Xinje XDPPro project, PLC1: XD3-32 (software 3.7.14 2021-12-24)

PROGRAM 梯形图

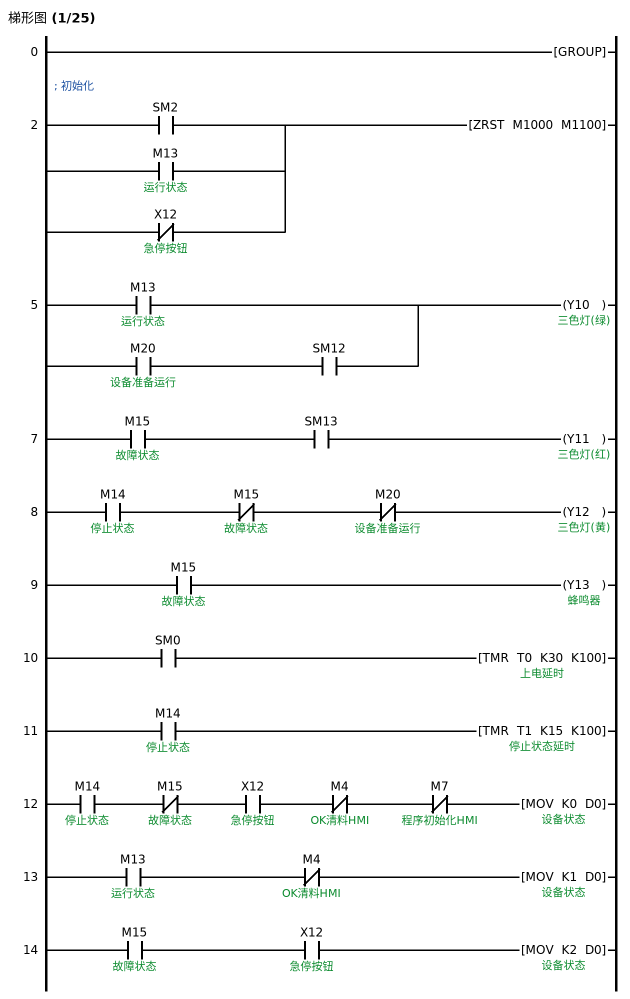
GROUP
; 初始化
LD     SM2
OR     M13	; 运行状态
ORI    X12	; 急停按钮
ZRST   M1000 M1100
LD     M13	; 运行状态
LD     M20	; 设备准备运行
AND    SM12
ORB
OUT    Y10	; 三色灯(绿)
LD     M15	; 故障状态
AND    SM13
OUT    Y11	; 三色灯(红)
LD     M14	; 停止状态
ANI    M15	; 故障状态
ANI    M20	; 设备准备运行
OUT    Y12	; 三色灯(黄)
LD     M15	; 故障状态
OUT    Y13	; 蜂鸣器
LD     SM0
TMR    T0 K30 K100	; 上电延时
LD     M14	; 停止状态
TMR    T1 K15 K100	; 停止状态延时
LD     M14	; 停止状态
ANI    M15	; 故障状态
AND    X12	; 急停按钮
ANI    M4	; OK清料HMI
ANI    M7	; 程序初始化HMI
MOV    K0 D0	; 设备状态
LD     M13	; 运行状态
ANI    M4	; OK清料HMI
MOV    K1 D0	; 设备状态
LD     M15	; 故障状态
AND    X12	; 急停按钮
MOV    K2 D0	; 设备状态

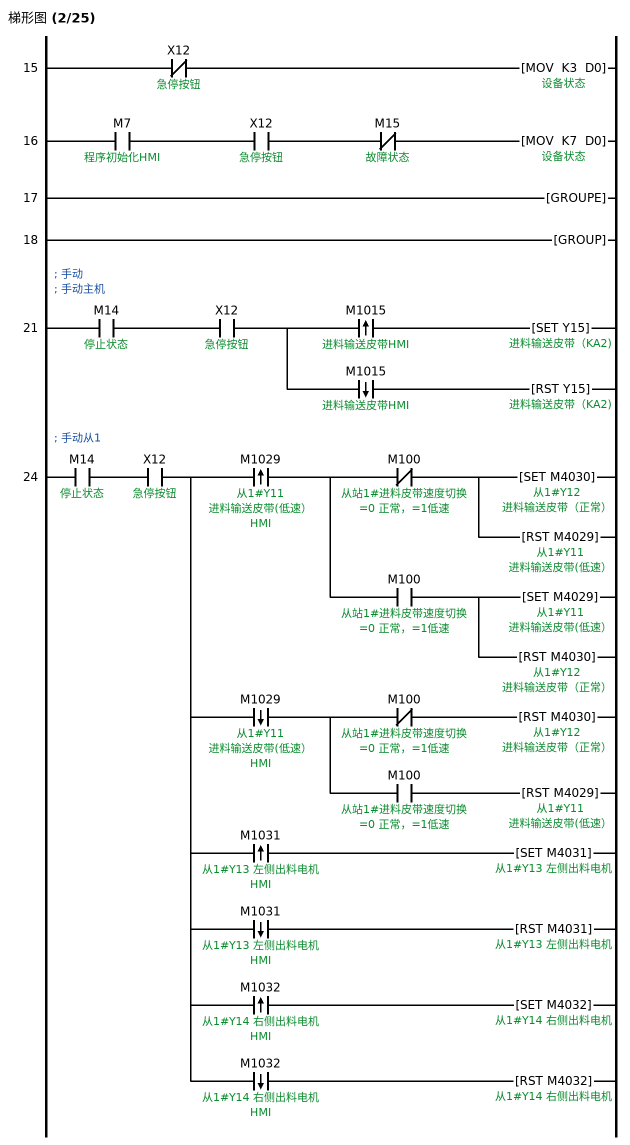
LDI    X12	; 急停按钮
MOV    K3 D0	; 设备状态
LD     M7	; 程序初始化HMI
AND    X12	; 急停按钮
ANI    M15	; 故障状态
MOV    K7 D0	; 设备状态
GROUPE
GROUP
; 手动
; 手动主机
LD     M14	; 停止状态
AND    X12	; 急停按钮
MPS
ANDP   M1015	; 进料输送皮带HMI
SET    Y15	; 进料输送皮带（KA2)
MPP
ANDF   M1015	; 进料输送皮带HMI
RST    Y15	; 进料输送皮带（KA2)
; 手动从1
LD     M14	; 停止状态
AND    X12	; 急停按钮
MPS
ANDP   M1029	; 从1#Y11 进料输送皮带(低速）       HMI
MPS
ANI    M100	; 从站1#进料皮带速度切换=0 正常，=1低速
SET    M4030	; 从1#Y12 进料输送皮带（正常）
RST    M4029	; 从1#Y11 进料输送皮带(低速）
MPP
AND    M100	; 从站1#进料皮带速度切换=0 正常，=1低速
SET    M4029	; 从1#Y11 进料输送皮带(低速）
RST    M4030	; 从1#Y12 进料输送皮带（正常）
MRD
ANDF   M1029	; 从1#Y11 进料输送皮带(低速）       HMI
MPS
ANI    M100	; 从站1#进料皮带速度切换=0 正常，=1低速
RST    M4030	; 从1#Y12 进料输送皮带（正常）
MPP
AND    M100	; 从站1#进料皮带速度切换=0 正常，=1低速
RST    M4029	; 从1#Y11 进料输送皮带(低速）
MRD
ANDP   M1031	; 从1#Y13 左侧出料电机       HMI
SET    M4031	; 从1#Y13 左侧出料电机
MRD
ANDF   M1031	; 从1#Y13 左侧出料电机       HMI
RST    M4031	; 从1#Y13 左侧出料电机
MRD
ANDP   M1032	; 从1#Y14 右侧出料电机       HMI
SET    M4032	; 从1#Y14 右侧出料电机
MPP
ANDF   M1032	; 从1#Y14 右侧出料电机       HMI
RST    M4032	; 从1#Y14 右侧出料电机

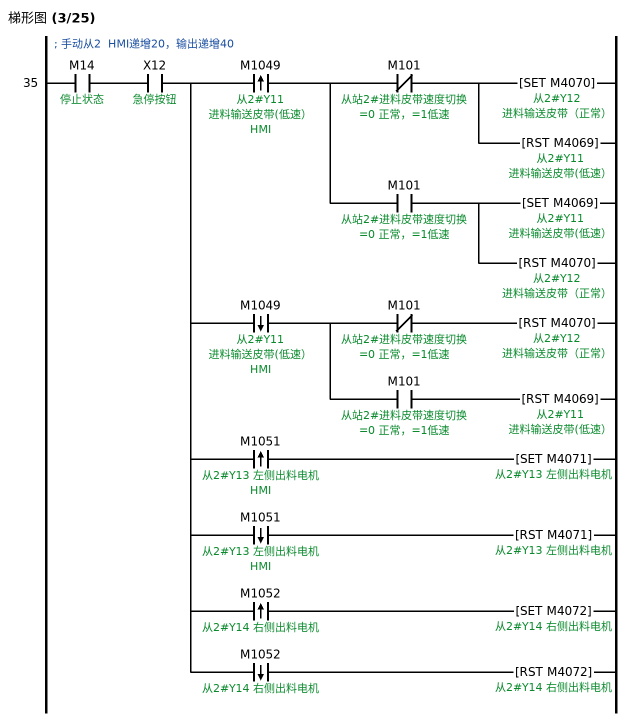
; 手动从2  HMI递增20，输出递增40
LD     M14	; 停止状态
AND    X12	; 急停按钮
MPS
ANDP   M1049	; 从2#Y11 进料输送皮带(低速）       HMI
MPS
ANI    M101	; 从站2#进料皮带速度切换=0 正常，=1低速
SET    M4070	; 从2#Y12 进料输送皮带（正常）
RST    M4069	; 从2#Y11 进料输送皮带(低速）
MPP
AND    M101	; 从站2#进料皮带速度切换=0 正常，=1低速
SET    M4069	; 从2#Y11 进料输送皮带(低速）
RST    M4070	; 从2#Y12 进料输送皮带（正常）
MRD
ANDF   M1049	; 从2#Y11 进料输送皮带(低速）       HMI
MPS
ANI    M101	; 从站2#进料皮带速度切换=0 正常，=1低速
RST    M4070	; 从2#Y12 进料输送皮带（正常）
MPP
AND    M101	; 从站2#进料皮带速度切换=0 正常，=1低速
RST    M4069	; 从2#Y11 进料输送皮带(低速）
MRD
ANDP   M1051	; 从2#Y13 左侧出料电机       HMI
SET    M4071	; 从2#Y13 左侧出料电机
MRD
ANDF   M1051	; 从2#Y13 左侧出料电机       HMI
RST    M4071	; 从2#Y13 左侧出料电机
MRD
ANDP   M1052	; 从2#Y14 右侧出料电机
SET    M4072	; 从2#Y14 右侧出料电机
MPP
ANDF   M1052	; 从2#Y14 右侧出料电机
RST    M4072	; 从2#Y14 右侧出料电机

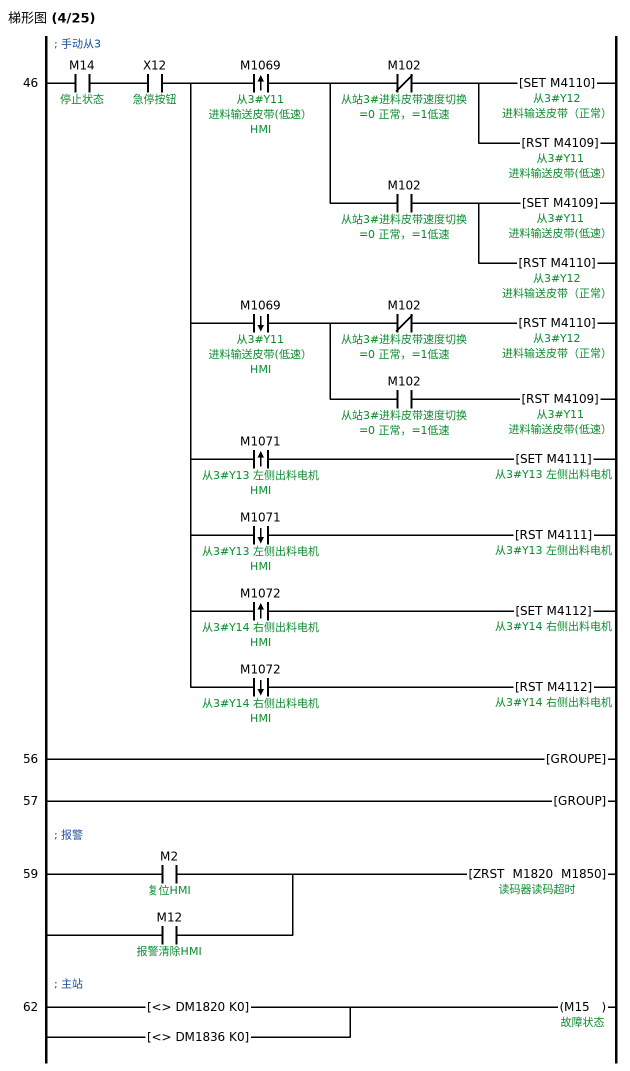
; 手动从3
LD     M14	; 停止状态
AND    X12	; 急停按钮
MPS
ANDP   M1069	; 从3#Y11 进料输送皮带(低速）       HMI
MPS
ANI    M102	; 从站3#进料皮带速度切换=0 正常，=1低速
SET    M4110	; 从3#Y12 进料输送皮带（正常）
RST    M4109	; 从3#Y11 进料输送皮带(低速）
MPP
AND    M102	; 从站3#进料皮带速度切换=0 正常，=1低速
SET    M4109	; 从3#Y11 进料输送皮带(低速）
RST    M4110	; 从3#Y12 进料输送皮带（正常）
MRD
ANDF   M1069	; 从3#Y11 进料输送皮带(低速）       HMI
MPS
ANI    M102	; 从站3#进料皮带速度切换=0 正常，=1低速
RST    M4110	; 从3#Y12 进料输送皮带（正常）
MPP
AND    M102	; 从站3#进料皮带速度切换=0 正常，=1低速
RST    M4109	; 从3#Y11 进料输送皮带(低速）
MRD
ANDP   M1071	; 从3#Y13 左侧出料电机       HMI
SET    M4111	; 从3#Y13 左侧出料电机
MRD
ANDF   M1071	; 从3#Y13 左侧出料电机       HMI
RST    M4111	; 从3#Y13 左侧出料电机
MRD
ANDP   M1072	; 从3#Y14 右侧出料电机       HMI
SET    M4112	; 从3#Y14 右侧出料电机
MPP
ANDF   M1072	; 从3#Y14 右侧出料电机       HMI
RST    M4112	; 从3#Y14 右侧出料电机
GROUPE
GROUP
; 报警
LD     M2	; 复位HMI
OR     M12	; 报警清除HMI
ZRST   M1820 M1850	; 读码器读码超时
; 主站
LD<>   DM1820 K0
OR<>   DM1836 K0
OUT    M15	; 故障状态

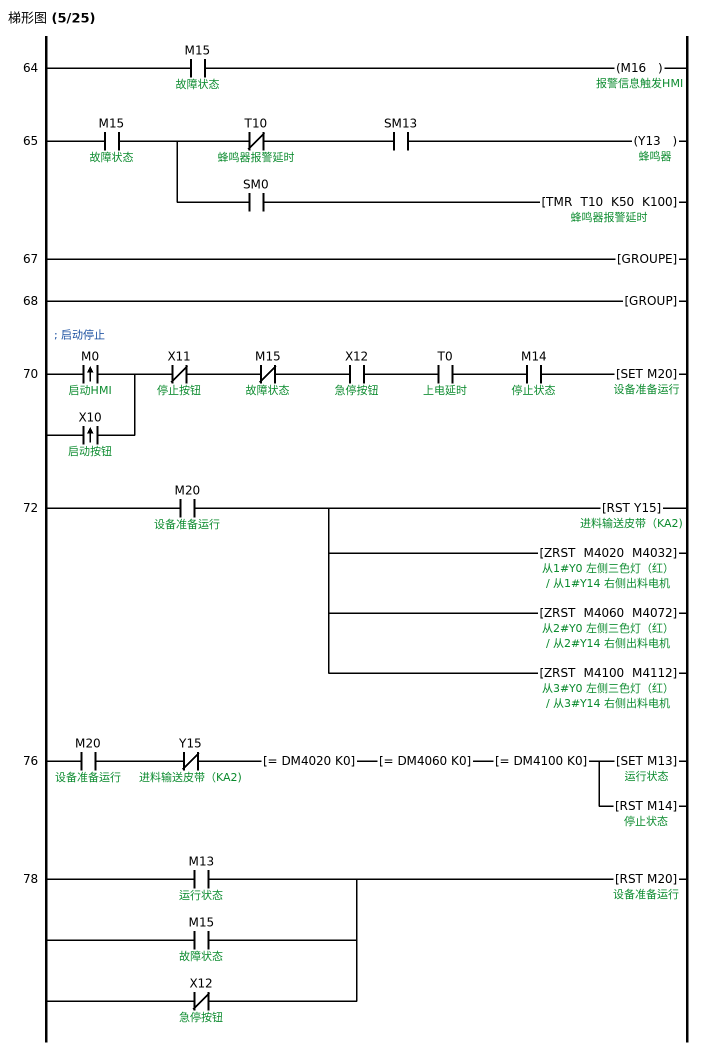
LD     M15	; 故障状态
OUT    M16	; 报警信息触发HMI
LD     M15	; 故障状态
MPS
ANI    T10	; 蜂鸣器报警延时
AND    SM13
OUT    Y13	; 蜂鸣器
MPP
AND    SM0
TMR    T10 K50 K100	; 蜂鸣器报警延时
GROUPE
GROUP
; 启动停止
LDP    M0	; 启动HMI
ORP    X10	; 启动按钮
ANI    X11	; 停止按钮
ANI    M15	; 故障状态
AND    X12	; 急停按钮
AND    T0	; 上电延时
AND    M14	; 停止状态
SET    M20	; 设备准备运行
LD     M20	; 设备准备运行
RST    Y15	; 进料输送皮带（KA2)
ZRST   M4020 M4032	; 从1#Y0 左侧三色灯（红） / 从1#Y14 右侧出料电机
ZRST   M4060 M4072	; 从2#Y0 左侧三色灯（红） / 从2#Y14 右侧出料电机
ZRST   M4100 M4112	; 从3#Y0 左侧三色灯（红） / 从3#Y14 右侧出料电机
LD     M20	; 设备准备运行
ANI    Y15	; 进料输送皮带（KA2)
AND=   DM4020 K0
AND=   DM4060 K0
AND=   DM4100 K0
SET    M13	; 运行状态
RST    M14	; 停止状态
LD     M13	; 运行状态
OR     M15	; 故障状态
ORI    X12	; 急停按钮
RST    M20	; 设备准备运行

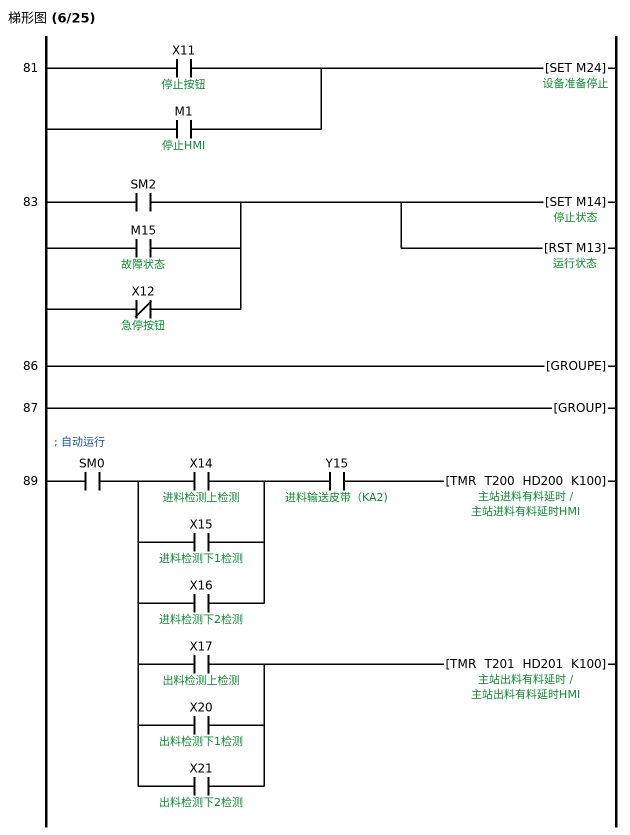
LD     X11	; 停止按钮
OR     M1	; 停止HMI
SET    M24	; 设备准备停止
LD     SM2
OR     M15	; 故障状态
ORI    X12	; 急停按钮
SET    M14	; 停止状态
RST    M13	; 运行状态
GROUPE
GROUP
; 自动运行
LD     SM0
MPS
LD     X14	; 进料检测上检测
OR     X15	; 进料检测下1检测
OR     X16	; 进料检测下2检测
ANB
AND    Y15	; 进料输送皮带（KA2)
TMR    T200 HD200 K100	; 主站进料有料延时 / 主站进料有料延时HMI
MPP
LD     X17	; 出料检测上检测
OR     X20	; 出料检测下1检测
OR     X21	; 出料检测下2检测
ANB
TMR    T201 HD201 K100	; 主站出料有料延时 / 主站出料有料延时HMI

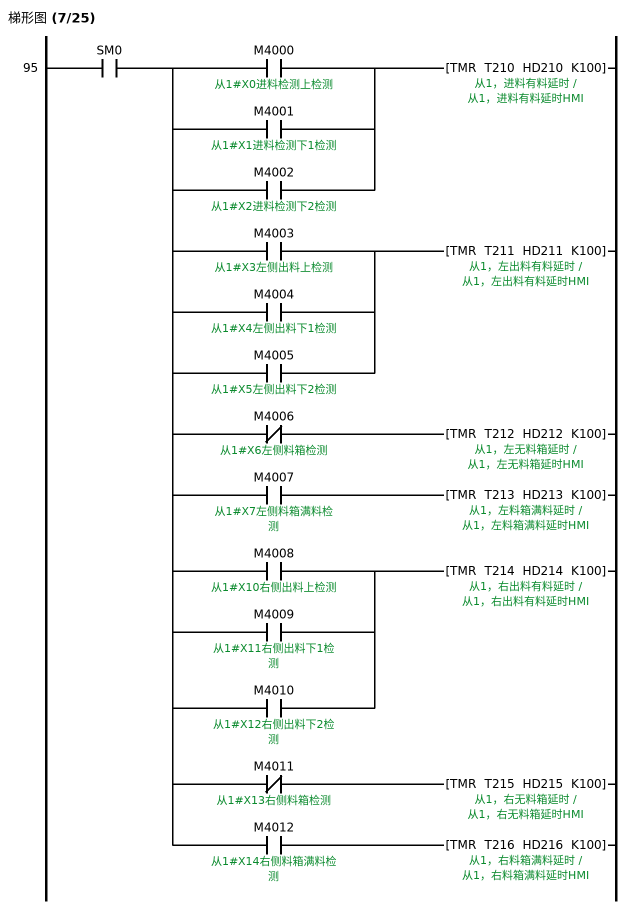
LD     SM0
MPS
LD     M4000	; 从1#X0进料检测上检测
OR     M4001	; 从1#X1进料检测下1检测
OR     M4002	; 从1#X2进料检测下2检测
ANB
TMR    T210 HD210 K100	; 从1，进料有料延时 / 从1，进料有料延时HMI
MRD
LD     M4003	; 从1#X3左侧出料上检测
OR     M4004	; 从1#X4左侧出料下1检测
OR     M4005	; 从1#X5左侧出料下2检测
ANB
TMR    T211 HD211 K100	; 从1，左出料有料延时 / 从1，左出料有料延时HMI
MRD
ANI    M4006	; 从1#X6左侧料箱检测
TMR    T212 HD212 K100	; 从1，左无料箱延时 / 从1，左无料箱延时HMI
MRD
AND    M4007	; 从1#X7左侧料箱满料检测
TMR    T213 HD213 K100	; 从1，左料箱满料延时 / 从1，左料箱满料延时HMI
MRD
LD     M4008	; 从1#X10右侧出料上检测
OR     M4009	; 从1#X11右侧出料下1检测
OR     M4010	; 从1#X12右侧出料下2检测
ANB
TMR    T214 HD214 K100	; 从1，右出料有料延时 / 从1，右出料有料延时HMI
MRD
ANI    M4011	; 从1#X13右侧料箱检测
TMR    T215 HD215 K100	; 从1，右无料箱延时 / 从1，右无料箱延时HMI
MPP
AND    M4012	; 从1#X14右侧料箱满料检测
TMR    T216 HD216 K100	; 从1，右料箱满料延时 / 从1，右料箱满料延时HMI

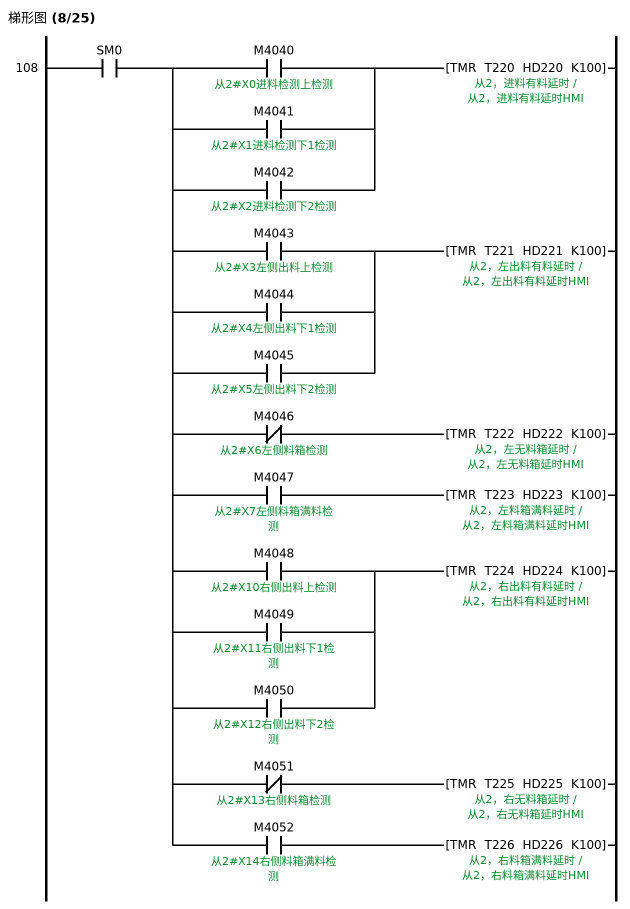
LD     SM0
MPS
LD     M4040	; 从2#X0进料检测上检测
OR     M4041	; 从2#X1进料检测下1检测
OR     M4042	; 从2#X2进料检测下2检测
ANB
TMR    T220 HD220 K100	; 从2，进料有料延时 / 从2，进料有料延时HMI
MRD
LD     M4043	; 从2#X3左侧出料上检测
OR     M4044	; 从2#X4左侧出料下1检测
OR     M4045	; 从2#X5左侧出料下2检测
ANB
TMR    T221 HD221 K100	; 从2，左出料有料延时 / 从2，左出料有料延时HMI
MRD
ANI    M4046	; 从2#X6左侧料箱检测
TMR    T222 HD222 K100	; 从2，左无料箱延时 / 从2，左无料箱延时HMI
MRD
AND    M4047	; 从2#X7左侧料箱满料检测
TMR    T223 HD223 K100	; 从2，左料箱满料延时 / 从2，左料箱满料延时HMI
MRD
LD     M4048	; 从2#X10右侧出料上检测
OR     M4049	; 从2#X11右侧出料下1检测
OR     M4050	; 从2#X12右侧出料下2检测
ANB
TMR    T224 HD224 K100	; 从2，右出料有料延时 / 从2，右出料有料延时HMI
MRD
ANI    M4051	; 从2#X13右侧料箱检测
TMR    T225 HD225 K100	; 从2，右无料箱延时 / 从2，右无料箱延时HMI
MPP
AND    M4052	; 从2#X14右侧料箱满料检测
TMR    T226 HD226 K100	; 从2，右料箱满料延时 / 从2，右料箱满料延时HMI

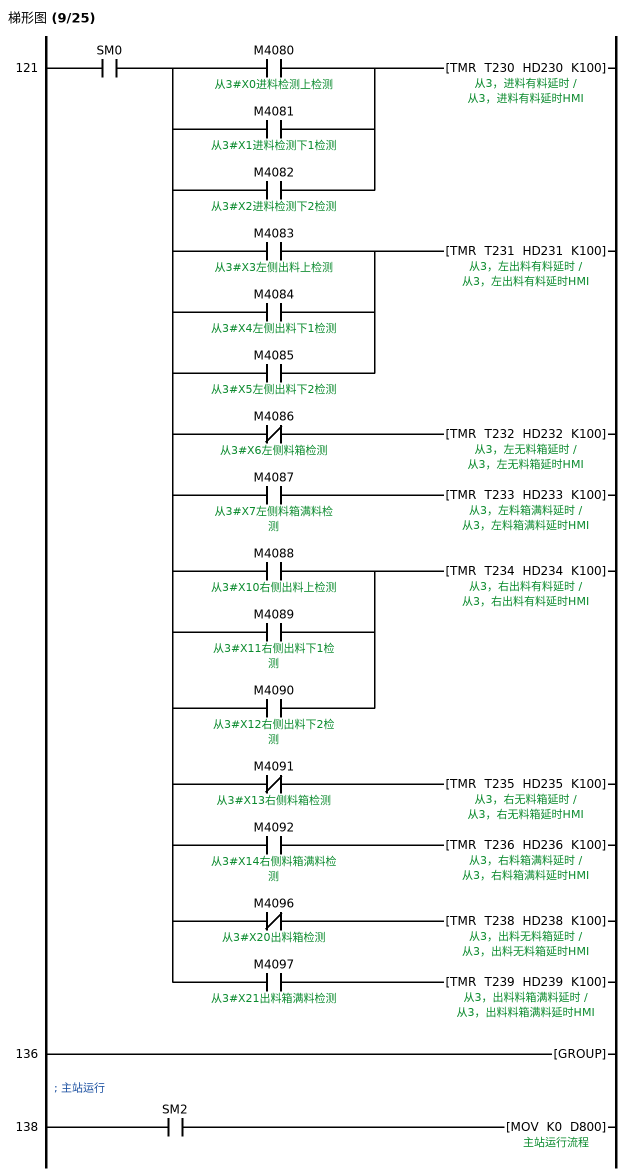
LD     SM0
MPS
LD     M4080	; 从3#X0进料检测上检测
OR     M4081	; 从3#X1进料检测下1检测
OR     M4082	; 从3#X2进料检测下2检测
ANB
TMR    T230 HD230 K100	; 从3，进料有料延时 / 从3，进料有料延时HMI
MRD
LD     M4083	; 从3#X3左侧出料上检测
OR     M4084	; 从3#X4左侧出料下1检测
OR     M4085	; 从3#X5左侧出料下2检测
ANB
TMR    T231 HD231 K100	; 从3，左出料有料延时 / 从3，左出料有料延时HMI
MRD
ANI    M4086	; 从3#X6左侧料箱检测
TMR    T232 HD232 K100	; 从3，左无料箱延时 / 从3，左无料箱延时HMI
MRD
AND    M4087	; 从3#X7左侧料箱满料检测
TMR    T233 HD233 K100	; 从3，左料箱满料延时 / 从3，左料箱满料延时HMI
MRD
LD     M4088	; 从3#X10右侧出料上检测
OR     M4089	; 从3#X11右侧出料下1检测
OR     M4090	; 从3#X12右侧出料下2检测
ANB
TMR    T234 HD234 K100	; 从3，右出料有料延时 / 从3，右出料有料延时HMI
MRD
ANI    M4091	; 从3#X13右侧料箱检测
TMR    T235 HD235 K100	; 从3，右无料箱延时 / 从3，右无料箱延时HMI
MRD
AND    M4092	; 从3#X14右侧料箱满料检测
TMR    T236 HD236 K100	; 从3，右料箱满料延时 / 从3，右料箱满料延时HMI
MRD
ANI    M4096	; 从3#X20出料箱检测
TMR    T238 HD238 K100	; 从3，出料无料箱延时 / 从3，出料无料箱延时HMI
MPP
AND    M4097	; 从3#X21出料箱满料检测
TMR    T239 HD239 K100	; 从3，出料料箱满料延时 / 从3，出料料箱满料延时HMI
GROUP
; 主站运行
LD     SM2
MOV    K0 D800	; 主站运行流程

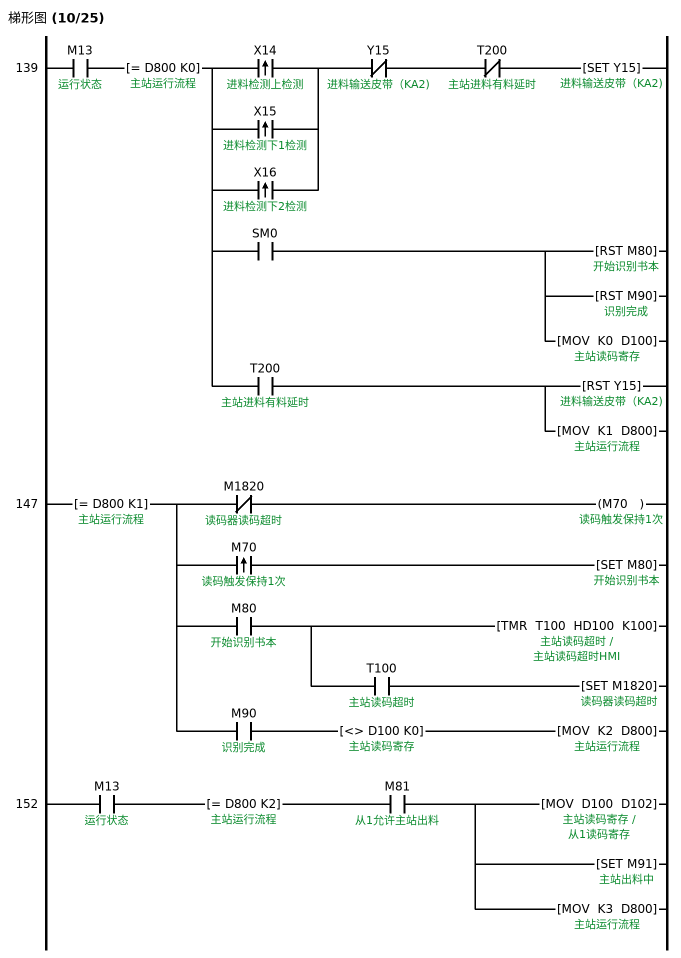
LD     M13	; 运行状态
AND=   D800 K0	; 主站运行流程
MPS
LDP    X14	; 进料检测上检测
ORP    X15	; 进料检测下1检测
ORP    X16	; 进料检测下2检测
ANB
ANI    Y15	; 进料输送皮带（KA2)
ANI    T200	; 主站进料有料延时
SET    Y15	; 进料输送皮带（KA2)
MRD
AND    SM0
RST    M80	; 开始识别书本
RST    M90	; 识别完成
MOV    K0 D100	; 主站读码寄存
MPP
AND    T200	; 主站进料有料延时
RST    Y15	; 进料输送皮带（KA2)
MOV    K1 D800	; 主站运行流程
LD=    D800 K1	; 主站运行流程
MPS
ANI    M1820	; 读码器读码超时
OUT    M70	; 读码触发保持1次
MRD
ANDP   M70	; 读码触发保持1次
SET    M80	; 开始识别书本
MRD
AND    M80	; 开始识别书本
TMR    T100 HD100 K100	; 主站读码超时 / 主站读码超时HMI
AND    T100	; 主站读码超时
SET    M1820	; 读码器读码超时
MPP
AND    M90	; 识别完成
AND<>  D100 K0	; 主站读码寄存
MOV    K2 D800	; 主站运行流程
LD     M13	; 运行状态
AND=   D800 K2	; 主站运行流程
AND    M81	; 从1允许主站出料
MOV    D100 D102	; 主站读码寄存 / 从1读码寄存
SET    M91	; 主站出料中
MOV    K3 D800	; 主站运行流程

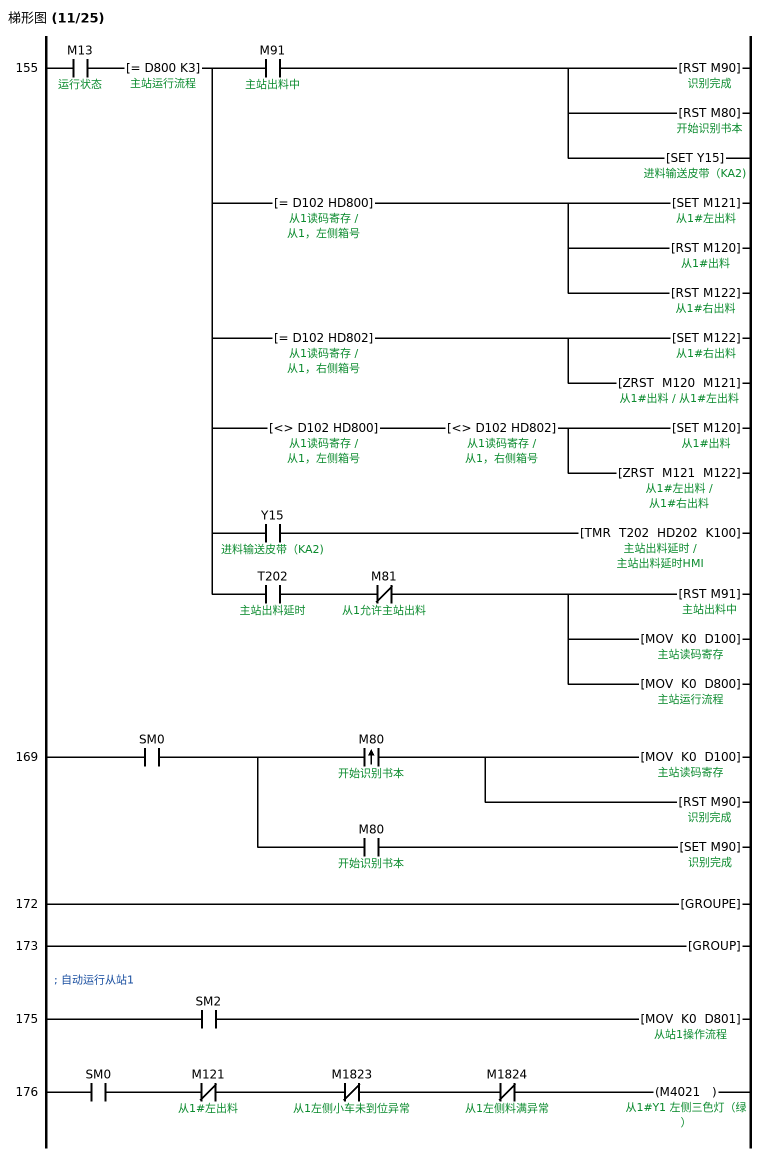
LD     M13	; 运行状态
AND=   D800 K3	; 主站运行流程
MPS
AND    M91	; 主站出料中
RST    M90	; 识别完成
RST    M80	; 开始识别书本
SET    Y15	; 进料输送皮带（KA2)
MRD
AND=   D102 HD800	; 从1读码寄存 / 从1，左侧箱号
SET    M121	; 从1#左出料
RST    M120	; 从1#出料
RST    M122	; 从1#右出料
MRD
AND=   D102 HD802	; 从1读码寄存 / 从1，右侧箱号
SET    M122	; 从1#右出料
ZRST   M120 M121	; 从1#出料 / 从1#左出料
MRD
AND<>  D102 HD800	; 从1读码寄存 / 从1，左侧箱号
AND<>  D102 HD802	; 从1读码寄存 / 从1，右侧箱号
SET    M120	; 从1#出料
ZRST   M121 M122	; 从1#左出料 / 从1#右出料
MRD
AND    Y15	; 进料输送皮带（KA2)
TMR    T202 HD202 K100	; 主站出料延时 / 主站出料延时HMI
MPP
AND    T202	; 主站出料延时
ANI    M81	; 从1允许主站出料
RST    M91	; 主站出料中
MOV    K0 D100	; 主站读码寄存
MOV    K0 D800	; 主站运行流程
LD     SM0
MPS
ANDP   M80	; 开始识别书本
MOV    K0 D100	; 主站读码寄存
RST    M90	; 识别完成
MPP
AND    M80	; 开始识别书本
SET    M90	; 识别完成
GROUPE
GROUP
; 自动运行从站1
LD     SM2
MOV    K0 D801	; 从站1操作流程
LD     SM0
ANI    M121	; 从1#左出料
ANI    M1823	; 从1左侧小车未到位异常
ANI    M1824	; 从1左侧料满异常
OUT    M4021	; 从1#Y1 左侧三色灯（绿）

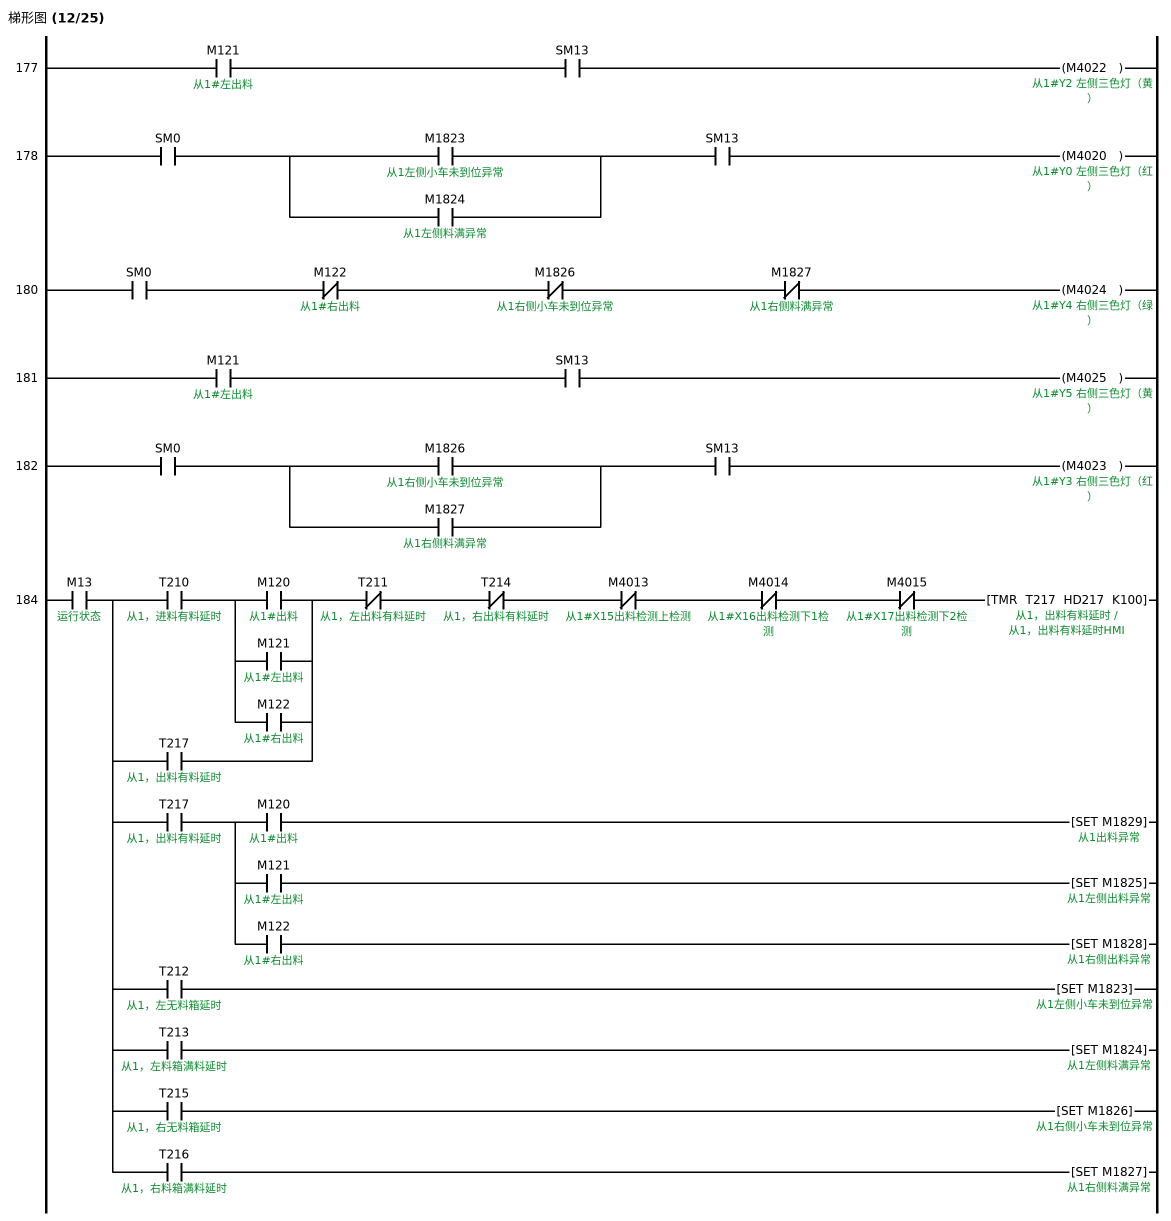
LD     M121	; 从1#左出料
AND    SM13
OUT    M4022	; 从1#Y2 左侧三色灯（黄）
LD     SM0
LD     M1823	; 从1左侧小车未到位异常
OR     M1824	; 从1左侧料满异常
ANB
AND    SM13
OUT    M4020	; 从1#Y0 左侧三色灯（红）
LD     SM0
ANI    M122	; 从1#右出料
ANI    M1826	; 从1右侧小车未到位异常
ANI    M1827	; 从1右侧料满异常
OUT    M4024	; 从1#Y4 右侧三色灯（绿）
LD     M121	; 从1#左出料
AND    SM13
OUT    M4025	; 从1#Y5 右侧三色灯（黄）
LD     SM0
LD     M1826	; 从1右侧小车未到位异常
OR     M1827	; 从1右侧料满异常
ANB
AND    SM13
OUT    M4023	; 从1#Y3 右侧三色灯（红）
LD     M13	; 运行状态
MPS
LD     T210	; 从1，进料有料延时
LD     M120	; 从1#出料
OR     M121	; 从1#左出料
OR     M122	; 从1#右出料
ANB
OR     T217	; 从1，出料有料延时
ANB
ANI    T211	; 从1，左出料有料延时
ANI    T214	; 从1，右出料有料延时
ANI    M4013	; 从1#X15出料检测上检测
ANI    M4014	; 从1#X16出料检测下1检测
ANI    M4015	; 从1#X17出料检测下2检测
TMR    T217 HD217 K100	; 从1，出料有料延时 / 从1，出料有料延时HMI
MRD
AND    T217	; 从1，出料有料延时
MPS
AND    M120	; 从1#出料
SET    M1829	; 从1出料异常
MRD
AND    M121	; 从1#左出料
SET    M1825	; 从1左侧出料异常
MPP
AND    M122	; 从1#右出料
SET    M1828	; 从1右侧出料异常
MRD
AND    T212	; 从1，左无料箱延时
SET    M1823	; 从1左侧小车未到位异常
MRD
AND    T213	; 从1，左料箱满料延时
SET    M1824	; 从1左侧料满异常
MRD
AND    T215	; 从1，右无料箱延时
SET    M1826	; 从1右侧小车未到位异常
MPP
AND    T216	; 从1，右料箱满料延时
SET    M1827	; 从1右侧料满异常

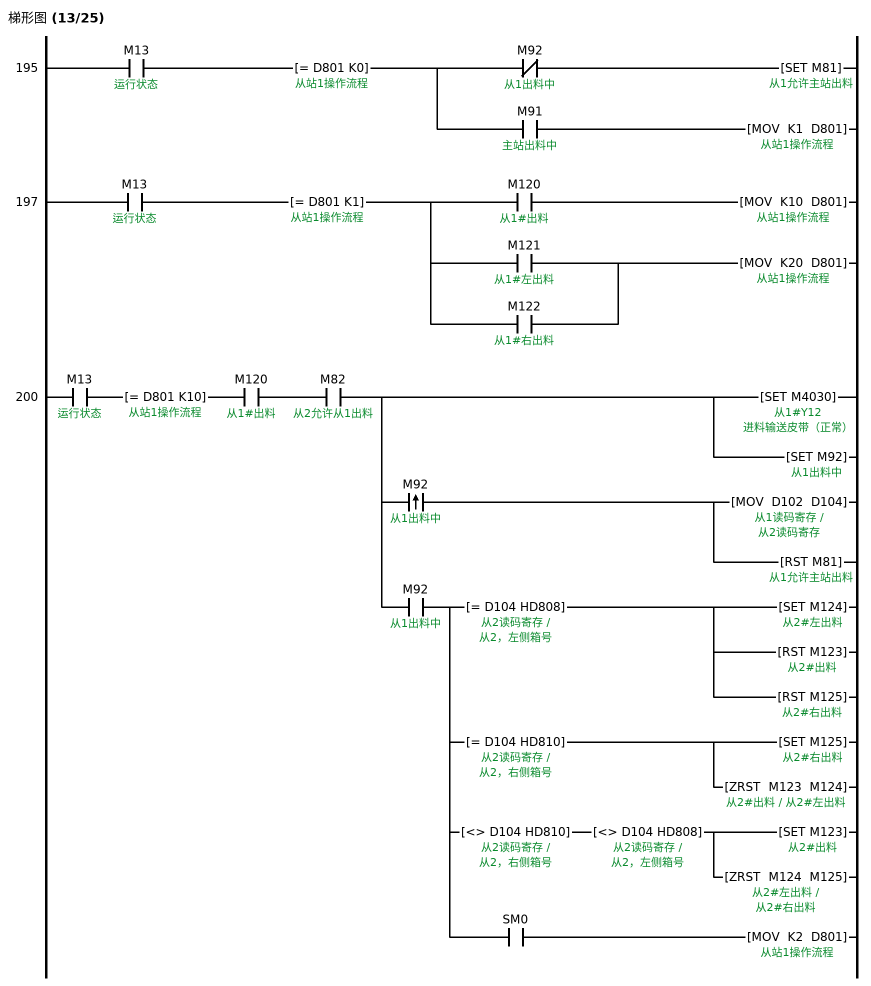
LD     M13	; 运行状态
AND=   D801 K0	; 从站1操作流程
MPS
ANI    M92	; 从1出料中
SET    M81	; 从1允许主站出料
MPP
AND    M91	; 主站出料中
MOV    K1 D801	; 从站1操作流程
LD     M13	; 运行状态
AND=   D801 K1	; 从站1操作流程
MPS
AND    M120	; 从1#出料
MOV    K10 D801	; 从站1操作流程
MPP
LD     M121	; 从1#左出料
OR     M122	; 从1#右出料
ANB
MOV    K20 D801	; 从站1操作流程
LD     M13	; 运行状态
AND=   D801 K10	; 从站1操作流程
AND    M120	; 从1#出料
AND    M82	; 从2允许从1出料
SET    M4030	; 从1#Y12 进料输送皮带（正常）
SET    M92	; 从1出料中
MPS
ANDP   M92	; 从1出料中
MOV    D102 D104	; 从1读码寄存 / 从2读码寄存
RST    M81	; 从1允许主站出料
MPP
AND    M92	; 从1出料中
MPS
AND=   D104 HD808	; 从2读码寄存 / 从2，左侧箱号
SET    M124	; 从2#左出料
RST    M123	; 从2#出料
RST    M125	; 从2#右出料
MRD
AND=   D104 HD810	; 从2读码寄存 / 从2，右侧箱号
SET    M125	; 从2#右出料
ZRST   M123 M124	; 从2#出料 / 从2#左出料
MRD
AND<>  D104 HD810	; 从2读码寄存 / 从2，右侧箱号
AND<>  D104 HD808	; 从2读码寄存 / 从2，左侧箱号
SET    M123	; 从2#出料
ZRST   M124 M125	; 从2#左出料 / 从2#右出料
MPP
AND    SM0
MOV    K2 D801	; 从站1操作流程

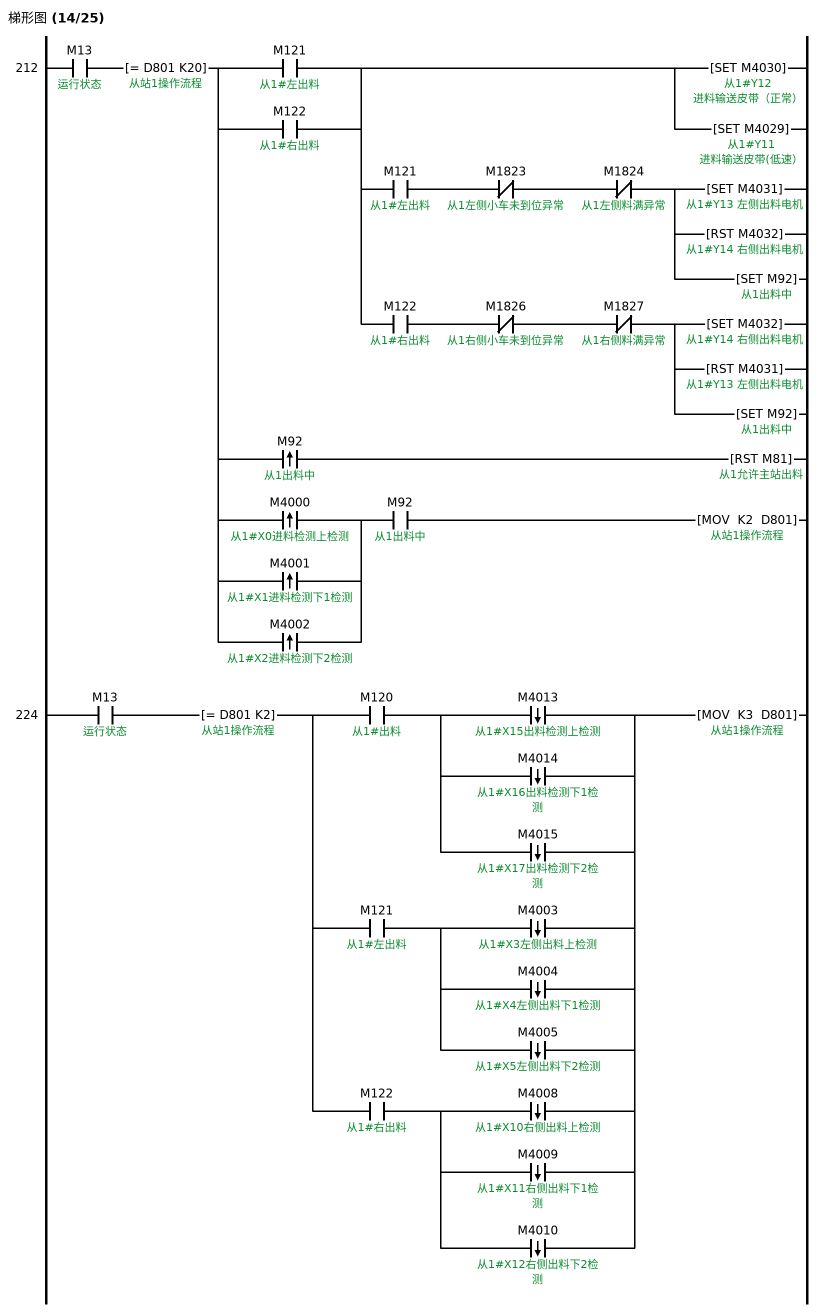
LD     M13	; 运行状态
AND=   D801 K20	; 从站1操作流程
MPS
LD     M121	; 从1#左出料
OR     M122	; 从1#右出料
ANB
SET    M4030	; 从1#Y12 进料输送皮带（正常）
SET    M4029	; 从1#Y11 进料输送皮带(低速）
MPS
AND    M121	; 从1#左出料
ANI    M1823	; 从1左侧小车未到位异常
ANI    M1824	; 从1左侧料满异常
SET    M4031	; 从1#Y13 左侧出料电机
RST    M4032	; 从1#Y14 右侧出料电机
SET    M92	; 从1出料中
MPP
AND    M122	; 从1#右出料
ANI    M1826	; 从1右侧小车未到位异常
ANI    M1827	; 从1右侧料满异常
SET    M4032	; 从1#Y14 右侧出料电机
RST    M4031	; 从1#Y13 左侧出料电机
SET    M92	; 从1出料中
MRD
ANDP   M92	; 从1出料中
RST    M81	; 从1允许主站出料
MPP
LDP    M4000	; 从1#X0进料检测上检测
ORP    M4001	; 从1#X1进料检测下1检测
ORP    M4002	; 从1#X2进料检测下2检测
ANB
AND    M92	; 从1出料中
MOV    K2 D801	; 从站1操作流程
LD     M13	; 运行状态
AND=   D801 K2	; 从站1操作流程
LD     M120	; 从1#出料
LDF    M4013	; 从1#X15出料检测上检测
ORF    M4014	; 从1#X16出料检测下1检测
ORF    M4015	; 从1#X17出料检测下2检测
ANB
LD     M121	; 从1#左出料
LDF    M4003	; 从1#X3左侧出料上检测
ORF    M4004	; 从1#X4左侧出料下1检测
ORF    M4005	; 从1#X5左侧出料下2检测
ANB
ORB
LD     M122	; 从1#右出料
LDF    M4008	; 从1#X10右侧出料上检测
ORF    M4009	; 从1#X11右侧出料下1检测
ORF    M4010	; 从1#X12右侧出料下2检测
ANB
ORB
ANB
MOV    K3 D801	; 从站1操作流程

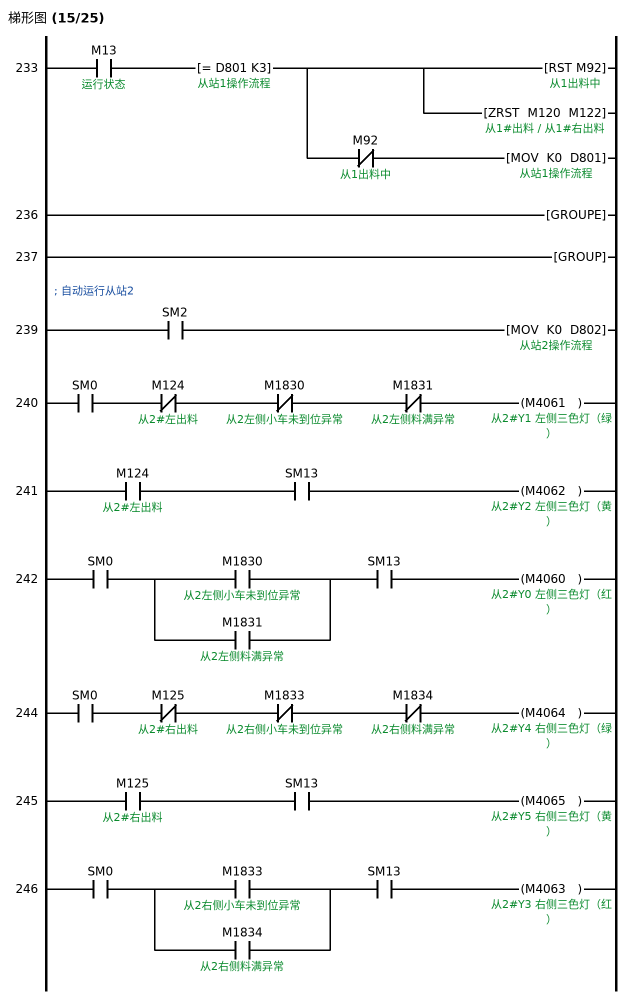
LD     M13	; 运行状态
AND=   D801 K3	; 从站1操作流程
RST    M92	; 从1出料中
ZRST   M120 M122	; 从1#出料 / 从1#右出料
ANI    M92	; 从1出料中
MOV    K0 D801	; 从站1操作流程
GROUPE
GROUP
; 自动运行从站2
LD     SM2
MOV    K0 D802	; 从站2操作流程
LD     SM0
ANI    M124	; 从2#左出料
ANI    M1830	; 从2左侧小车未到位异常
ANI    M1831	; 从2左侧料满异常
OUT    M4061	; 从2#Y1 左侧三色灯（绿）
LD     M124	; 从2#左出料
AND    SM13
OUT    M4062	; 从2#Y2 左侧三色灯（黄）
LD     SM0
LD     M1830	; 从2左侧小车未到位异常
OR     M1831	; 从2左侧料满异常
ANB
AND    SM13
OUT    M4060	; 从2#Y0 左侧三色灯（红）
LD     SM0
ANI    M125	; 从2#右出料
ANI    M1833	; 从2右侧小车未到位异常
ANI    M1834	; 从2右侧料满异常
OUT    M4064	; 从2#Y4 右侧三色灯（绿）
LD     M125	; 从2#右出料
AND    SM13
OUT    M4065	; 从2#Y5 右侧三色灯（黄）
LD     SM0
LD     M1833	; 从2右侧小车未到位异常
OR     M1834	; 从2右侧料满异常
ANB
AND    SM13
OUT    M4063	; 从2#Y3 右侧三色灯（红）

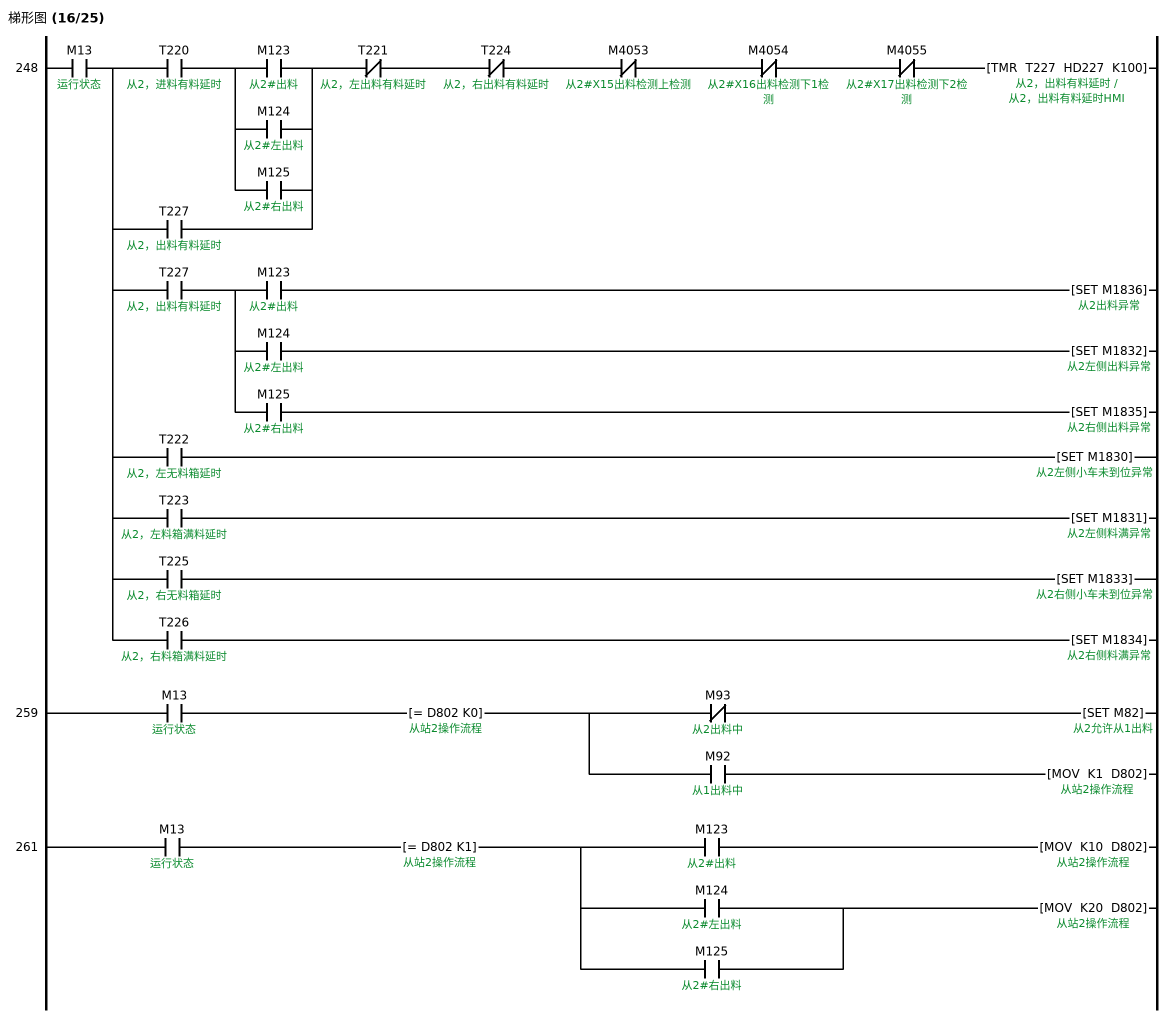
LD     M13	; 运行状态
MPS
LD     T220	; 从2，进料有料延时
LD     M123	; 从2#出料
OR     M124	; 从2#左出料
OR     M125	; 从2#右出料
ANB
OR     T227	; 从2，出料有料延时
ANB
ANI    T221	; 从2，左出料有料延时
ANI    T224	; 从2，右出料有料延时
ANI    M4053	; 从2#X15出料检测上检测
ANI    M4054	; 从2#X16出料检测下1检测
ANI    M4055	; 从2#X17出料检测下2检测
TMR    T227 HD227 K100	; 从2，出料有料延时 / 从2，出料有料延时HMI
MRD
AND    T227	; 从2，出料有料延时
MPS
AND    M123	; 从2#出料
SET    M1836	; 从2出料异常
MRD
AND    M124	; 从2#左出料
SET    M1832	; 从2左侧出料异常
MPP
AND    M125	; 从2#右出料
SET    M1835	; 从2右侧出料异常
MRD
AND    T222	; 从2，左无料箱延时
SET    M1830	; 从2左侧小车未到位异常
MRD
AND    T223	; 从2，左料箱满料延时
SET    M1831	; 从2左侧料满异常
MRD
AND    T225	; 从2，右无料箱延时
SET    M1833	; 从2右侧小车未到位异常
MPP
AND    T226	; 从2，右料箱满料延时
SET    M1834	; 从2右侧料满异常
LD     M13	; 运行状态
AND=   D802 K0	; 从站2操作流程
MPS
ANI    M93	; 从2出料中
SET    M82	; 从2允许从1出料
MPP
AND    M92	; 从1出料中
MOV    K1 D802	; 从站2操作流程
LD     M13	; 运行状态
AND=   D802 K1	; 从站2操作流程
MPS
AND    M123	; 从2#出料
MOV    K10 D802	; 从站2操作流程
MPP
LD     M124	; 从2#左出料
OR     M125	; 从2#右出料
ANB
MOV    K20 D802	; 从站2操作流程

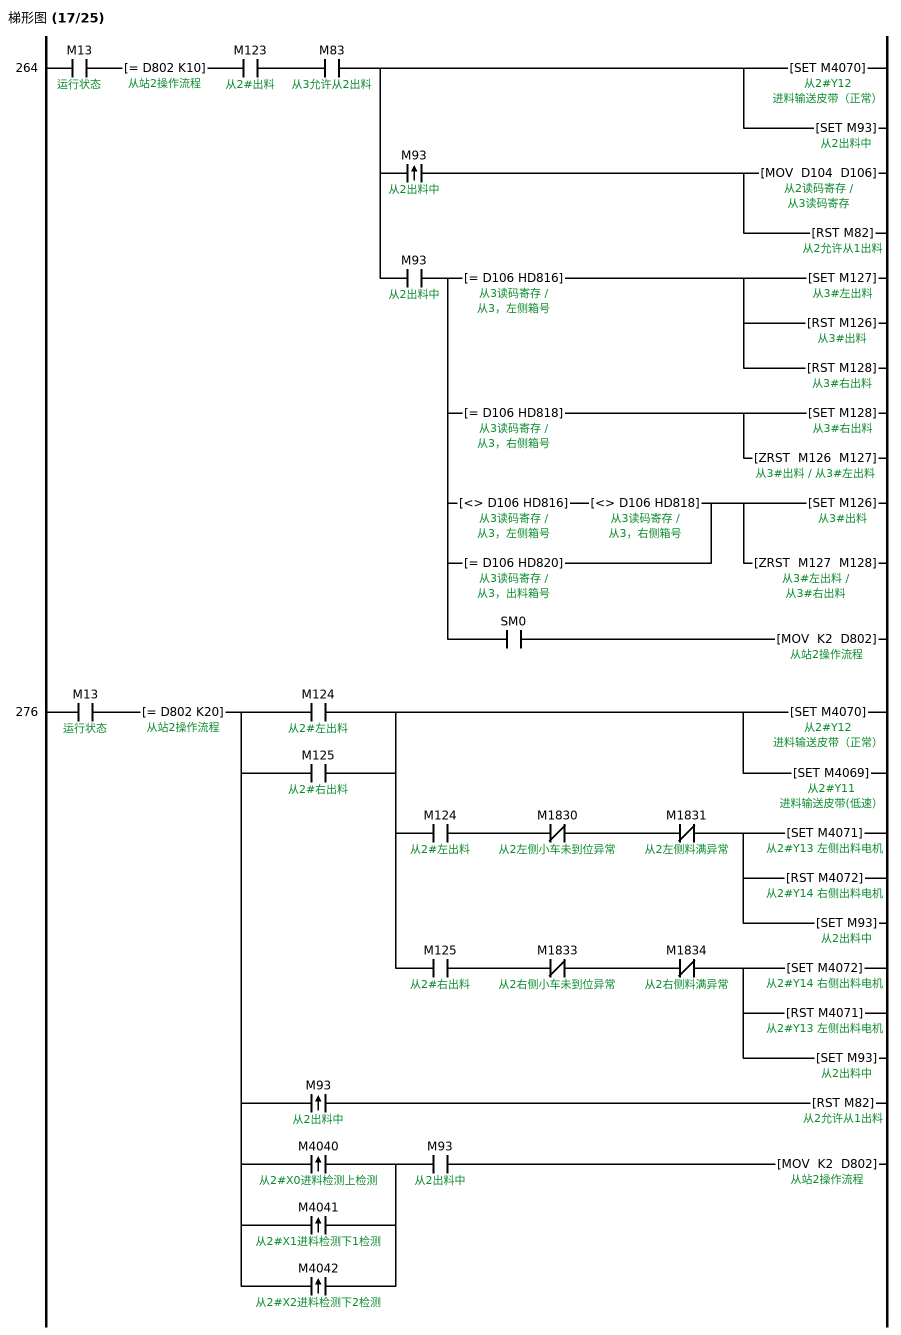
LD     M13	; 运行状态
AND=   D802 K10	; 从站2操作流程
AND    M123	; 从2#出料
AND    M83	; 从3允许从2出料
SET    M4070	; 从2#Y12 进料输送皮带（正常）
SET    M93	; 从2出料中
MPS
ANDP   M93	; 从2出料中
MOV    D104 D106	; 从2读码寄存 / 从3读码寄存
RST    M82	; 从2允许从1出料
MPP
AND    M93	; 从2出料中
MPS
AND=   D106 HD816	; 从3读码寄存 / 从3，左侧箱号
SET    M127	; 从3#左出料
RST    M126	; 从3#出料
RST    M128	; 从3#右出料
MRD
AND=   D106 HD818	; 从3读码寄存 / 从3，右侧箱号
SET    M128	; 从3#右出料
ZRST   M126 M127	; 从3#出料 / 从3#左出料
MRD
LD<>   D106 HD816	; 从3读码寄存 / 从3，左侧箱号
AND<>  D106 HD818	; 从3读码寄存 / 从3，右侧箱号
OR=    D106 HD820	; 从3读码寄存 / 从3，出料箱号
ANB
SET    M126	; 从3#出料
ZRST   M127 M128	; 从3#左出料 / 从3#右出料
MPP
AND    SM0
MOV    K2 D802	; 从站2操作流程
LD     M13	; 运行状态
AND=   D802 K20	; 从站2操作流程
MPS
LD     M124	; 从2#左出料
OR     M125	; 从2#右出料
ANB
SET    M4070	; 从2#Y12 进料输送皮带（正常）
SET    M4069	; 从2#Y11 进料输送皮带(低速）
MPS
AND    M124	; 从2#左出料
ANI    M1830	; 从2左侧小车未到位异常
ANI    M1831	; 从2左侧料满异常
SET    M4071	; 从2#Y13 左侧出料电机
RST    M4072	; 从2#Y14 右侧出料电机
SET    M93	; 从2出料中
MPP
AND    M125	; 从2#右出料
ANI    M1833	; 从2右侧小车未到位异常
ANI    M1834	; 从2右侧料满异常
SET    M4072	; 从2#Y14 右侧出料电机
RST    M4071	; 从2#Y13 左侧出料电机
SET    M93	; 从2出料中
MRD
ANDP   M93	; 从2出料中
RST    M82	; 从2允许从1出料
MPP
LDP    M4040	; 从2#X0进料检测上检测
ORP    M4041	; 从2#X1进料检测下1检测
ORP    M4042	; 从2#X2进料检测下2检测
ANB
AND    M93	; 从2出料中
MOV    K2 D802	; 从站2操作流程

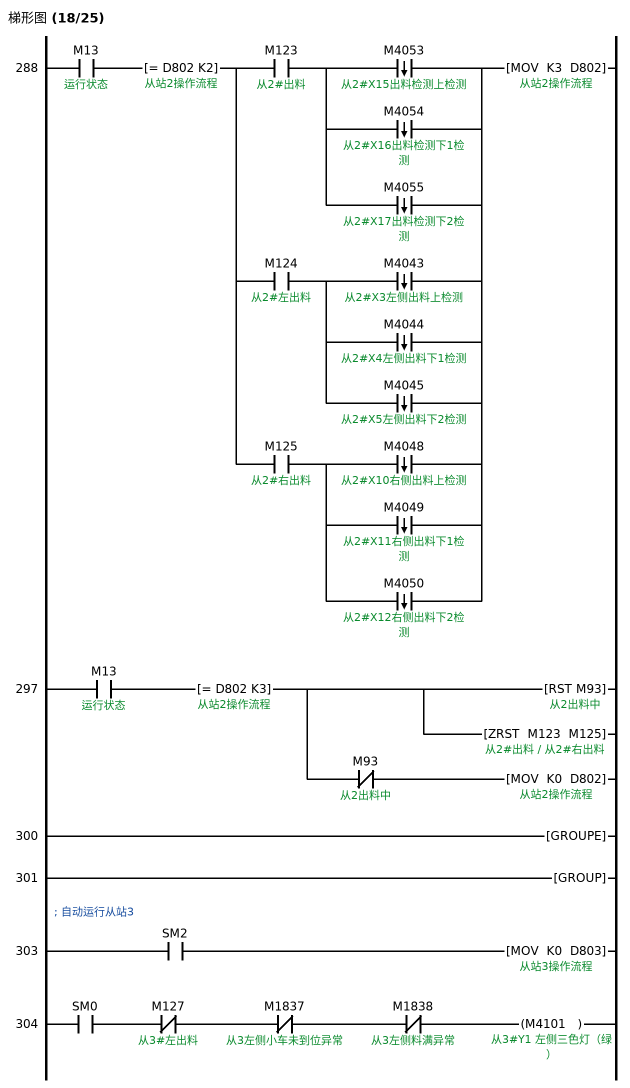
LD     M13	; 运行状态
AND=   D802 K2	; 从站2操作流程
LD     M123	; 从2#出料
LDF    M4053	; 从2#X15出料检测上检测
ORF    M4054	; 从2#X16出料检测下1检测
ORF    M4055	; 从2#X17出料检测下2检测
ANB
LD     M124	; 从2#左出料
LDF    M4043	; 从2#X3左侧出料上检测
ORF    M4044	; 从2#X4左侧出料下1检测
ORF    M4045	; 从2#X5左侧出料下2检测
ANB
ORB
LD     M125	; 从2#右出料
LDF    M4048	; 从2#X10右侧出料上检测
ORF    M4049	; 从2#X11右侧出料下1检测
ORF    M4050	; 从2#X12右侧出料下2检测
ANB
ORB
ANB
MOV    K3 D802	; 从站2操作流程
LD     M13	; 运行状态
AND=   D802 K3	; 从站2操作流程
RST    M93	; 从2出料中
ZRST   M123 M125	; 从2#出料 / 从2#右出料
ANI    M93	; 从2出料中
MOV    K0 D802	; 从站2操作流程
GROUPE
GROUP
; 自动运行从站3
LD     SM2
MOV    K0 D803	; 从站3操作流程
LD     SM0
ANI    M127	; 从3#左出料
ANI    M1837	; 从3左侧小车未到位异常
ANI    M1838	; 从3左侧料满异常
OUT    M4101	; 从3#Y1 左侧三色灯（绿）

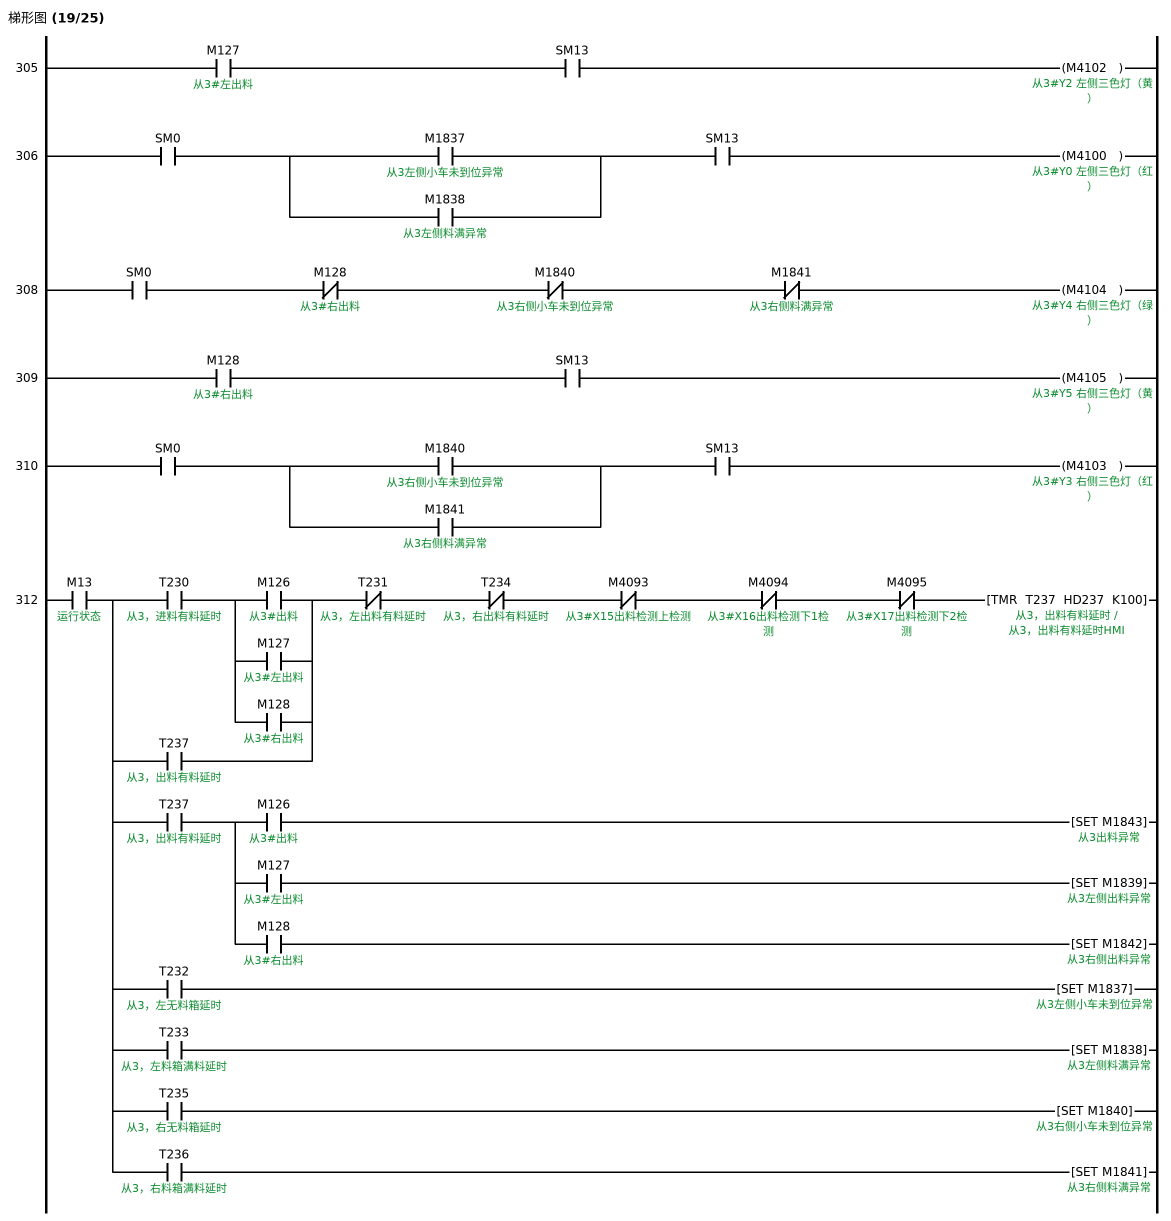
LD     M127	; 从3#左出料
AND    SM13
OUT    M4102	; 从3#Y2 左侧三色灯（黄）
LD     SM0
LD     M1837	; 从3左侧小车未到位异常
OR     M1838	; 从3左侧料满异常
ANB
AND    SM13
OUT    M4100	; 从3#Y0 左侧三色灯（红）
LD     SM0
ANI    M128	; 从3#右出料
ANI    M1840	; 从3右侧小车未到位异常
ANI    M1841	; 从3右侧料满异常
OUT    M4104	; 从3#Y4 右侧三色灯（绿）
LD     M128	; 从3#右出料
AND    SM13
OUT    M4105	; 从3#Y5 右侧三色灯（黄）
LD     SM0
LD     M1840	; 从3右侧小车未到位异常
OR     M1841	; 从3右侧料满异常
ANB
AND    SM13
OUT    M4103	; 从3#Y3 右侧三色灯（红）
LD     M13	; 运行状态
MPS
LD     T230	; 从3，进料有料延时
LD     M126	; 从3#出料
OR     M127	; 从3#左出料
OR     M128	; 从3#右出料
ANB
OR     T237	; 从3，出料有料延时
ANB
ANI    T231	; 从3，左出料有料延时
ANI    T234	; 从3，右出料有料延时
ANI    M4093	; 从3#X15出料检测上检测
ANI    M4094	; 从3#X16出料检测下1检测
ANI    M4095	; 从3#X17出料检测下2检测
TMR    T237 HD237 K100	; 从3，出料有料延时 / 从3，出料有料延时HMI
MRD
AND    T237	; 从3，出料有料延时
MPS
AND    M126	; 从3#出料
SET    M1843	; 从3出料异常
MRD
AND    M127	; 从3#左出料
SET    M1839	; 从3左侧出料异常
MPP
AND    M128	; 从3#右出料
SET    M1842	; 从3右侧出料异常
MRD
AND    T232	; 从3，左无料箱延时
SET    M1837	; 从3左侧小车未到位异常
MRD
AND    T233	; 从3，左料箱满料延时
SET    M1838	; 从3左侧料满异常
MRD
AND    T235	; 从3，右无料箱延时
SET    M1840	; 从3右侧小车未到位异常
MPP
AND    T236	; 从3，右料箱满料延时
SET    M1841	; 从3右侧料满异常

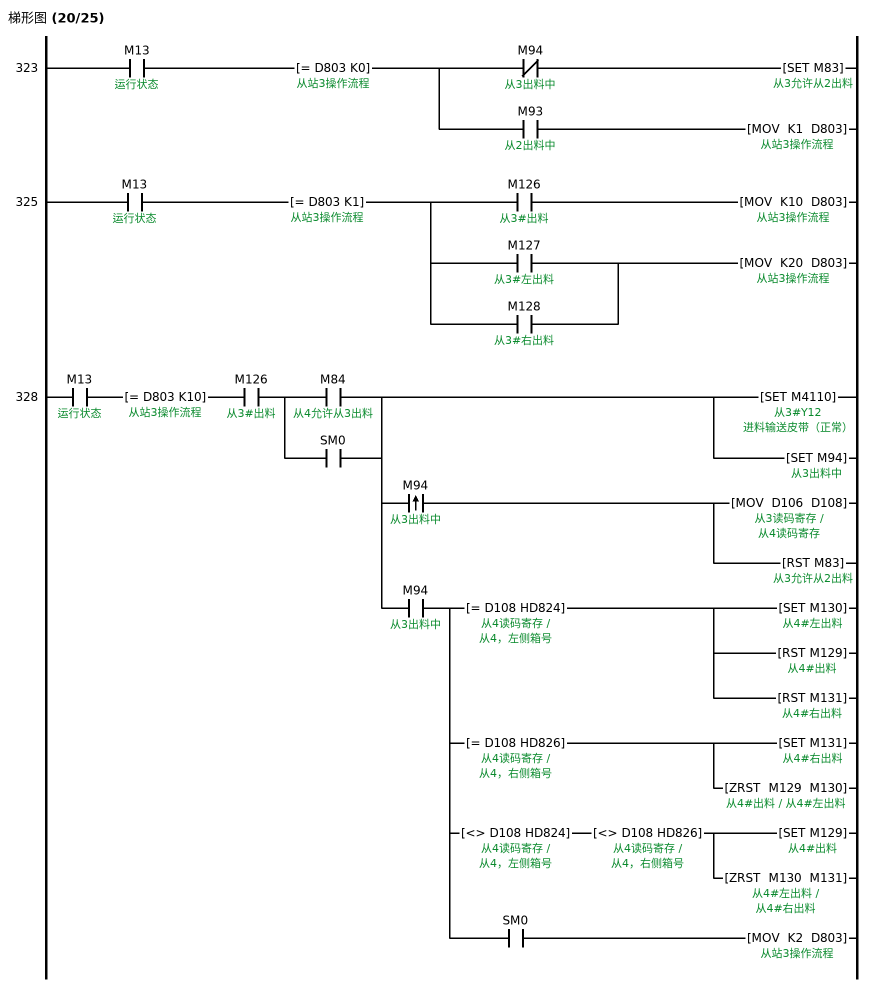
LD     M13	; 运行状态
AND=   D803 K0	; 从站3操作流程
MPS
ANI    M94	; 从3出料中
SET    M83	; 从3允许从2出料
MPP
AND    M93	; 从2出料中
MOV    K1 D803	; 从站3操作流程
LD     M13	; 运行状态
AND=   D803 K1	; 从站3操作流程
MPS
AND    M126	; 从3#出料
MOV    K10 D803	; 从站3操作流程
MPP
LD     M127	; 从3#左出料
OR     M128	; 从3#右出料
ANB
MOV    K20 D803	; 从站3操作流程
LD     M13	; 运行状态
AND=   D803 K10	; 从站3操作流程
AND    M126	; 从3#出料
LD     M84	; 从4允许从3出料
OR     SM0
ANB
SET    M4110	; 从3#Y12 进料输送皮带（正常）
SET    M94	; 从3出料中
MPS
ANDP   M94	; 从3出料中
MOV    D106 D108	; 从3读码寄存 / 从4读码寄存
RST    M83	; 从3允许从2出料
MPP
AND    M94	; 从3出料中
MPS
AND=   D108 HD824	; 从4读码寄存 / 从4，左侧箱号
SET    M130	; 从4#左出料
RST    M129	; 从4#出料
RST    M131	; 从4#右出料
MRD
AND=   D108 HD826	; 从4读码寄存 / 从4，右侧箱号
SET    M131	; 从4#右出料
ZRST   M129 M130	; 从4#出料 / 从4#左出料
MRD
AND<>  D108 HD824	; 从4读码寄存 / 从4，左侧箱号
AND<>  D108 HD826	; 从4读码寄存 / 从4，右侧箱号
SET    M129	; 从4#出料
ZRST   M130 M131	; 从4#左出料 / 从4#右出料
MPP
AND    SM0
MOV    K2 D803	; 从站3操作流程

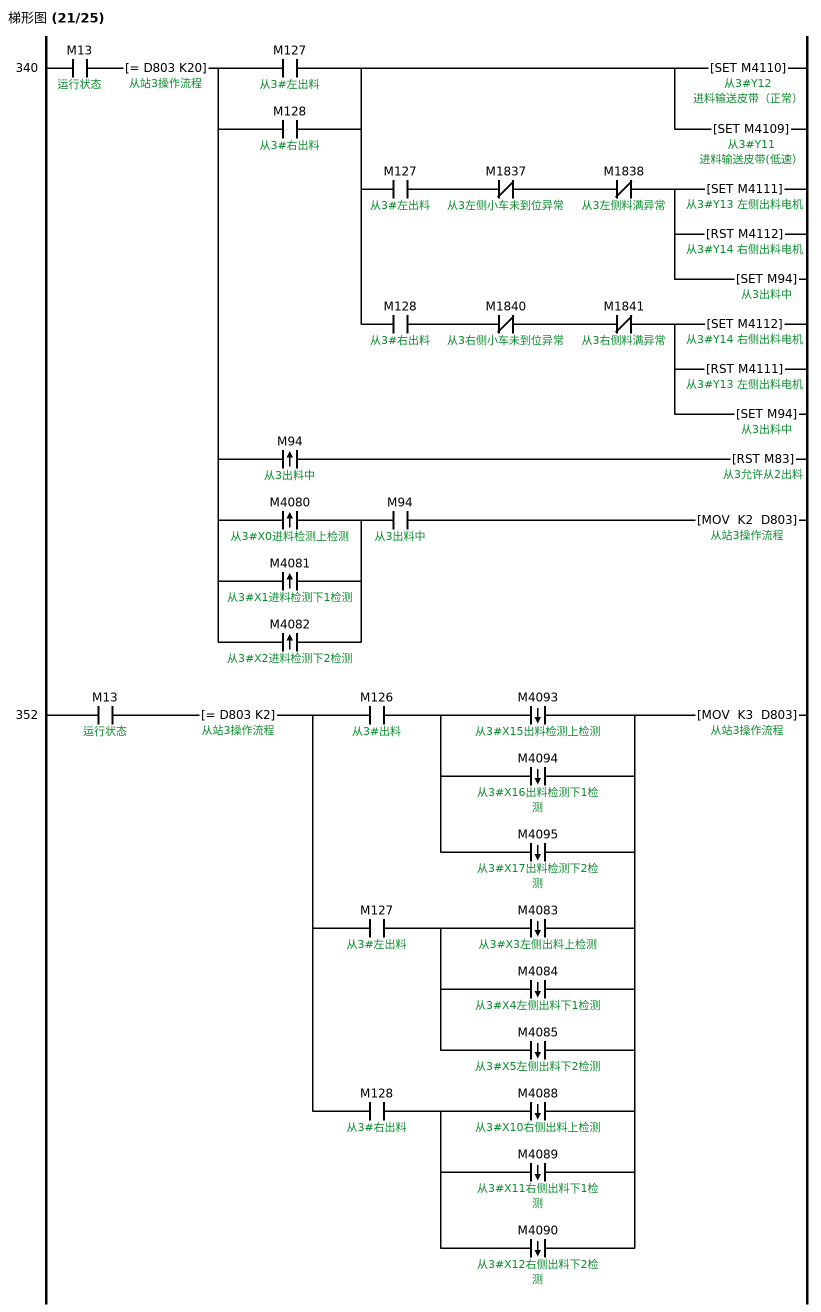
LD     M13	; 运行状态
AND=   D803 K20	; 从站3操作流程
MPS
LD     M127	; 从3#左出料
OR     M128	; 从3#右出料
ANB
SET    M4110	; 从3#Y12 进料输送皮带（正常）
SET    M4109	; 从3#Y11 进料输送皮带(低速）
MPS
AND    M127	; 从3#左出料
ANI    M1837	; 从3左侧小车未到位异常
ANI    M1838	; 从3左侧料满异常
SET    M4111	; 从3#Y13 左侧出料电机
RST    M4112	; 从3#Y14 右侧出料电机
SET    M94	; 从3出料中
MPP
AND    M128	; 从3#右出料
ANI    M1840	; 从3右侧小车未到位异常
ANI    M1841	; 从3右侧料满异常
SET    M4112	; 从3#Y14 右侧出料电机
RST    M4111	; 从3#Y13 左侧出料电机
SET    M94	; 从3出料中
MRD
ANDP   M94	; 从3出料中
RST    M83	; 从3允许从2出料
MPP
LDP    M4080	; 从3#X0进料检测上检测
ORP    M4081	; 从3#X1进料检测下1检测
ORP    M4082	; 从3#X2进料检测下2检测
ANB
AND    M94	; 从3出料中
MOV    K2 D803	; 从站3操作流程
LD     M13	; 运行状态
AND=   D803 K2	; 从站3操作流程
LD     M126	; 从3#出料
LDF    M4093	; 从3#X15出料检测上检测
ORF    M4094	; 从3#X16出料检测下1检测
ORF    M4095	; 从3#X17出料检测下2检测
ANB
LD     M127	; 从3#左出料
LDF    M4083	; 从3#X3左侧出料上检测
ORF    M4084	; 从3#X4左侧出料下1检测
ORF    M4085	; 从3#X5左侧出料下2检测
ANB
ORB
LD     M128	; 从3#右出料
LDF    M4088	; 从3#X10右侧出料上检测
ORF    M4089	; 从3#X11右侧出料下1检测
ORF    M4090	; 从3#X12右侧出料下2检测
ANB
ORB
ANB
MOV    K3 D803	; 从站3操作流程

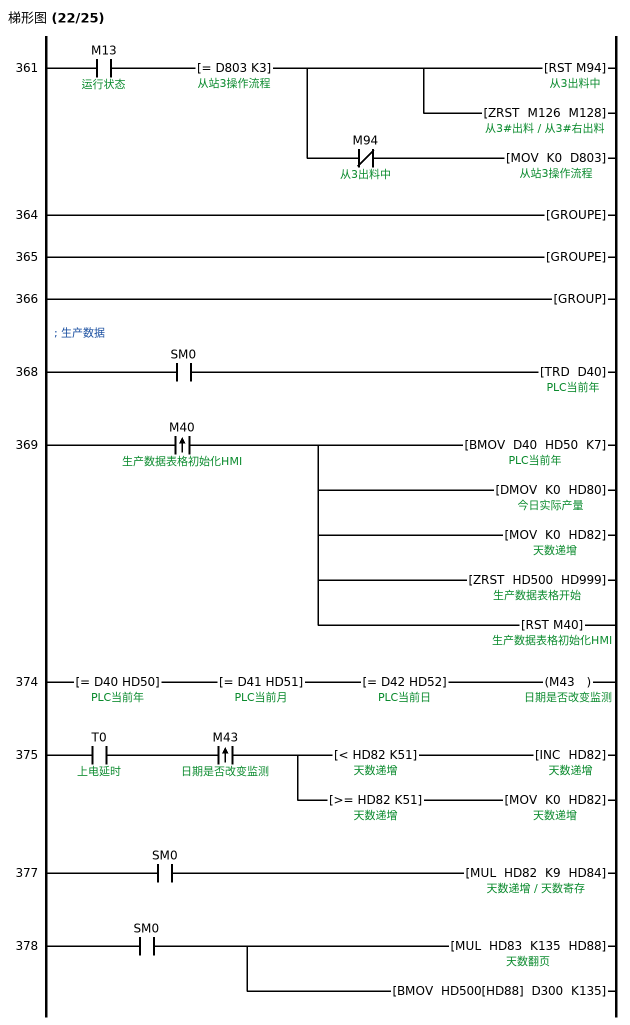
LD     M13	; 运行状态
AND=   D803 K3	; 从站3操作流程
RST    M94	; 从3出料中
ZRST   M126 M128	; 从3#出料 / 从3#右出料
ANI    M94	; 从3出料中
MOV    K0 D803	; 从站3操作流程
GROUPE
GROUPE
GROUP
; 生产数据
LD     SM0
TRD    D40	; PLC当前年
LDP    M40	; 生产数据表格初始化HMI
BMOV   D40 HD50 K7	; PLC当前年
DMOV   K0 HD80	; 今日实际产量
MOV    K0 HD82	; 天数递增
ZRST   HD500 HD999	; 生产数据表格开始
RST    M40	; 生产数据表格初始化HMI
LD=    D40 HD50	; PLC当前年
AND=   D41 HD51	; PLC当前月
AND=   D42 HD52	; PLC当前日
OUT    M43	; 日期是否改变监测
LD     T0	; 上电延时
ANDP   M43	; 日期是否改变监测
MPS
AND<   HD82 K51	; 天数递增
INC    HD82	; 天数递增
MPP
AND>=  HD82 K51	; 天数递增
MOV    K0 HD82	; 天数递增
LD     SM0
MUL    HD82 K9 HD84	; 天数递增 / 天数寄存
LD     SM0
MUL    HD83 K135 HD88	; 天数翻页
BMOV   HD500[HD88] D300 K135

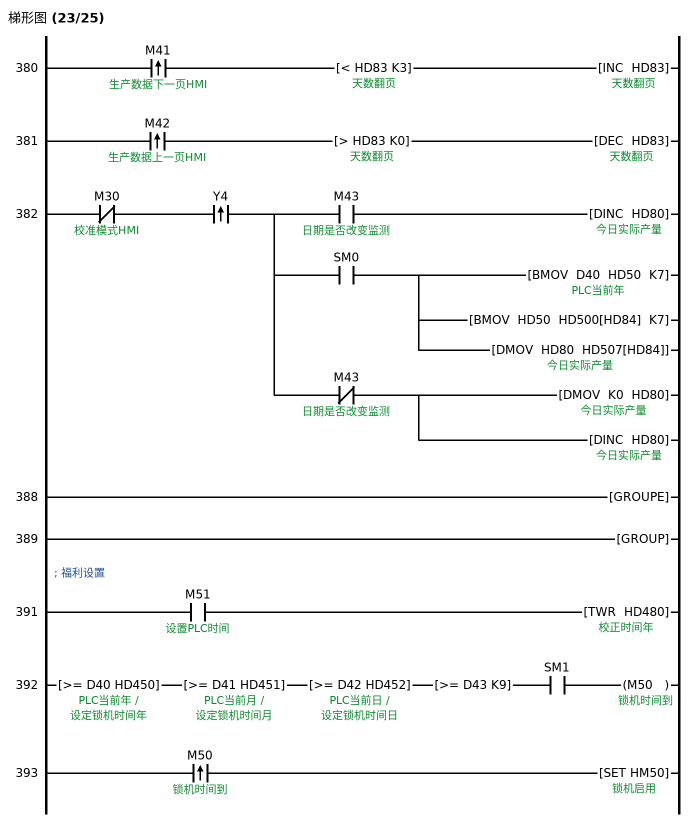
LDP    M41	; 生产数据下一页HMI
AND<   HD83 K3	; 天数翻页
INC    HD83	; 天数翻页
LDP    M42	; 生产数据上一页HMI
AND>   HD83 K0	; 天数翻页
DEC    HD83	; 天数翻页
LDI    M30	; 校准模式HMI
ANDP   Y4
MPS
AND    M43	; 日期是否改变监测
DINC   HD80	; 今日实际产量
MRD
AND    SM0
BMOV   D40 HD50 K7	; PLC当前年
BMOV   HD50 HD500[HD84] K7
DMOV   HD80 HD507[HD84]	; 今日实际产量
MPP
ANI    M43	; 日期是否改变监测
DMOV   K0 HD80	; 今日实际产量
DINC   HD80	; 今日实际产量
GROUPE
GROUP
; 福利设置
LD     M51	; 设置PLC时间
TWR    HD480	; 校正时间年
LD>=   D40 HD450	; PLC当前年 / 设定锁机时间年
AND>=  D41 HD451	; PLC当前月 / 设定锁机时间月
AND>=  D42 HD452	; PLC当前日 / 设定锁机时间日
AND>=  D43 K9
AND    SM1
OUT    M50	; 锁机时间到
LDP    M50	; 锁机时间到
SET    HM50	; 锁机启用

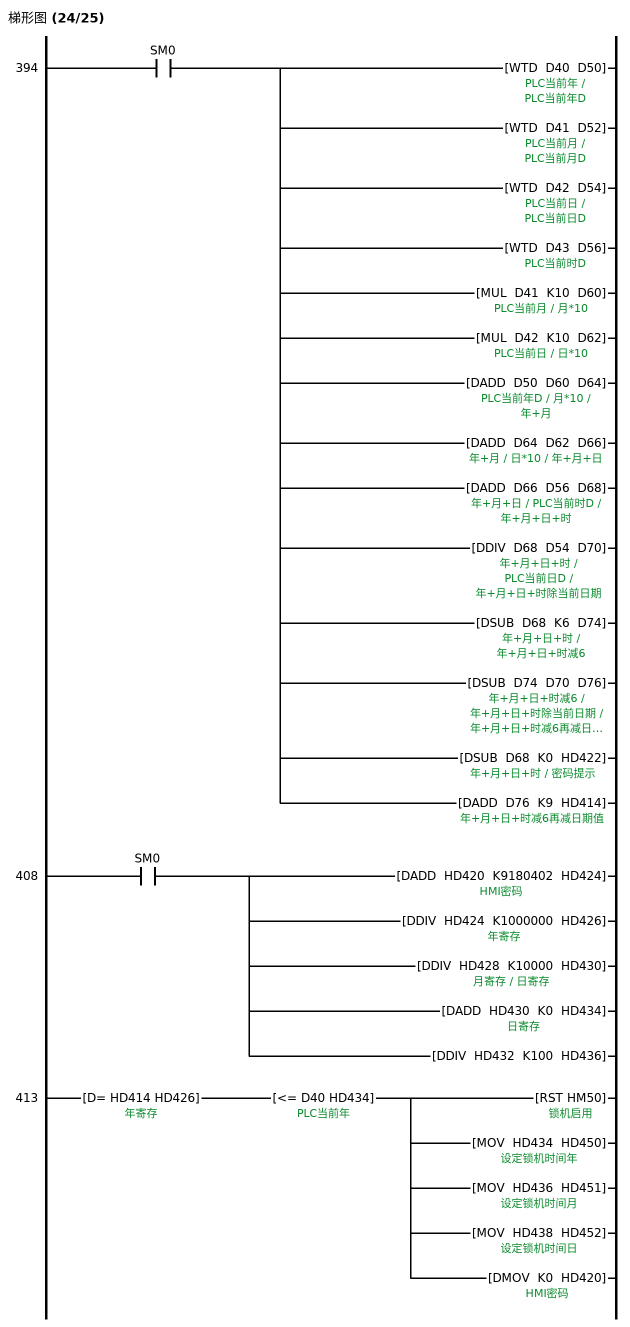
LD     SM0
WTD    D40 D50	; PLC当前年 / PLC当前年D
WTD    D41 D52	; PLC当前月 / PLC当前月D
WTD    D42 D54	; PLC当前日 / PLC当前日D
WTD    D43 D56	; PLC当前时D
MUL    D41 K10 D60	; PLC当前月 / 月*10
MUL    D42 K10 D62	; PLC当前日 / 日*10
DADD   D50 D60 D64	; PLC当前年D / 月*10 / 年+月
DADD   D64 D62 D66	; 年+月 / 日*10 / 年+月+日
DADD   D66 D56 D68	; 年+月+日 / PLC当前时D / 年+月+日+时
DDIV   D68 D54 D70	; 年+月+日+时 / PLC当前日D / 年+月+日+时除当前日期
DSUB   D68 K6 D74	; 年+月+日+时 / 年+月+日+时减6
DSUB   D74 D70 D76	; 年+月+日+时减6 / 年+月+日+时除当前日期 / 年+月+日+时减6再减日期值
DSUB   D68 K0 HD422	; 年+月+日+时 / 密码提示
DADD   D76 K9 HD414	; 年+月+日+时减6再减日期值
LD     SM0
DADD   HD420 K9180402 HD424	; HMI密码
DDIV   HD424 K1000000 HD426	; 年寄存
DDIV   HD428 K10000 HD430	; 月寄存 / 日寄存
DADD   HD430 K0 HD434	; 日寄存
DDIV   HD432 K100 HD436
DLD=   HD414 HD426	; 年寄存
AND<=  D40 HD434	; PLC当前年
RST    HM50	; 锁机启用
MOV    HD434 HD450	; 设定锁机时间年
MOV    HD436 HD451	; 设定锁机时间月
MOV    HD438 HD452	; 设定锁机时间日
DMOV   K0 HD420	; HMI密码

